(* CoDeSys 2.3.9.41 project: advance.pro *)
(* Libraries: UNM.lib 14.2.06 12:27:08, SmsOwenLib.lib 5.10.12 16:48:36, STANDARD.LIB 4.10.05 10:14:46, IECSFC.LIB 13.4.06 14:51:28, SYSLIBTIME.LIB 20.2.06 13:31:16, SYSTASKINFO.LIB 20.2.06 13:31:38, ANALYZATION.LIB 5.10.99 08:05:06, SYSLIBCALLBACK.LIB 20.2.06 13:31:08 *)

(* PLC configuration (modules and I/O channels)
Discrete input 8 bit [ID100] node 0, in %IB0 out %QB0 {Filtrationtime = 10; Filtrationtime = 10; Filtrationtime = 10; Filtrationtime = 10; Filtrationtime = 10; Filtrationtime = 10; Filtrationtime = 10; Filtrationtime = 10; Visibility = No; PinCount = 8; WatchDogPeriod = 1000; PollPeriod = 1}
  AT %IB0.0 [ByteInput] 8 discrete inputs
Discrete output 2 bit [ID101] node 1, in %IB1 out %QB1 {PinCount = 2; SafeValueBool = FALSE; SafeValueBool = FALSE; Visibility = No}
  pmp1 AT %QX1.0 [BitOutput] First
  pmp2 AT %QX1.1 [BitOutput] Second
Discrete output 2 bit [ID101] node 2, in %IB2 out %QB2 {PinCount = 2; SafeValueBool = FALSE; SafeValueBool = FALSE; Visibility = No}
  pmp3 AT %QX2.0 [BitOutput] First
  pmp4 AT %QX2.1 [BitOutput] Second
Discrete output 2 bit [ID101] node 3, in %IB3 out %QB3 {PinCount = 2; SafeValueBool = FALSE; SafeValueBool = FALSE; Visibility = No}
  AT %QX3.0 [BitOutput] First
  AT %QX3.1 [BitOutput] Second
Discrete output 2 bit [ID101] node 4, in %IB4 out %QB4 {PinCount = 2; SafeValueBool = FALSE; SafeValueBool = FALSE; Visibility = No}
  AT %QX4.0 [BitOutput] First
  AT %QX4.1 [BitOutput] Second
Discrete output 2 bit [ID101] node 5, in %IB5 out %QB5 {PinCount = 2; SafeValueBool = FALSE; SafeValueBool = FALSE; Visibility = No}
  AT %QX5.0 [BitOutput] First
  AT %QX5.1 [BitOutput] Second
Discrete output 2 bit [ID101] node 6, in %IB6 out %QB6 {PinCount = 2; SafeValueBool = FALSE; SafeValueBool = FALSE; Visibility = No}
  AT %QX6.0 [BitOutput] First
  AT %QX6.1 [BitOutput] Second
Special output [ID104] node 7, in %IB7 out %QB7 {Visibility = No; PinCount = 1}
  AT %QX7.0 [BitOutput] Special output
RS-232 [COM2_USART] node 0, in %IB8.0 out %QB8.0 {CommunicationSpeed = 9600; Parity = NO PARITY CHECK; BitLength = 8 bits; StopLength = One stop bit; InterfaceType = RS232; FrameOriented = ASCII; Timeout = 0; Visibility = No}
*)

(* Global variable list: Global_Variables *)
VAR_GLOBAL

	SMS_ID  : WORD;

END_VAR

(* POU PLC_PRG, ST *)
PROGRAM PLC_PRG
VAR
    startTimer, waitBeforeStartPmp2, waitBeforeStartPmp3, waitBeforeStartPmp4 : TON;
    letsGo : BOOL;
    letsStop : BOOL;
    stopTimer,waitBeforeStopPmp3,  waitBeforeStopPmp2, waitBeforeStopPmp1 : TON;
    startBreak, pmp2break, pmp3break, pmp4break : BOOL;

END_VAR
Process;

SMS;
END_PROGRAM
ACTION Process:
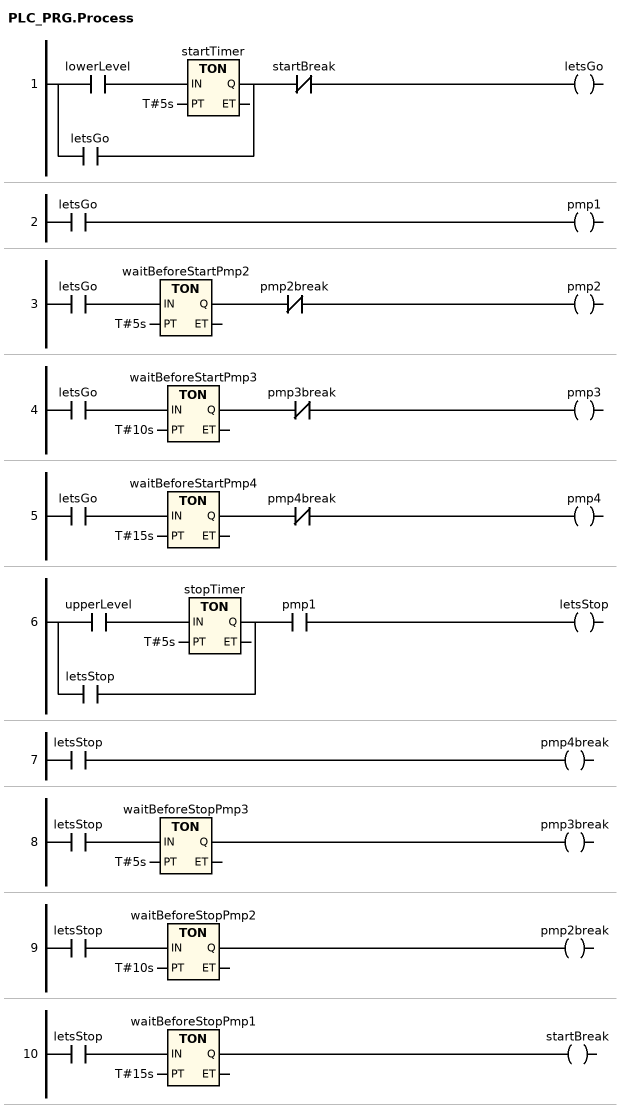
_LD_ (* Ladder Diagram *)
NETWORK 1
	{ [lowerLevel] - startTimer:TON(IN: *, PT: T#5s) | [letsGo] } - [/startBreak] --- (letsGo)
NETWORK 2
	[letsGo] --- (pmp1)
NETWORK 3
	[letsGo] - waitBeforeStartPmp2:TON(IN: *, PT: T#5s) - [/pmp2break] --- (pmp2)
NETWORK 4
	[letsGo] - waitBeforeStartPmp3:TON(IN: *, PT: T#10s) - [/pmp3break] --- (pmp3)
NETWORK 5
	[letsGo] - waitBeforeStartPmp4:TON(IN: *, PT: T#15s) - [/pmp4break] --- (pmp4)
NETWORK 6
	{ [upperLevel] - stopTimer:TON(IN: *, PT: T#5s) | [letsStop] } - [pmp1] --- (letsStop)
NETWORK 7
	[letsStop] --- (pmp4break)
NETWORK 8
	[letsStop] - waitBeforeStopPmp3:TON(IN: *, PT: T#5s) --- (pmp3break)
NETWORK 9
	[letsStop] - waitBeforeStopPmp2:TON(IN: *, PT: T#10s) --- (pmp2break)
NETWORK 10
	[letsStop] - waitBeforeStopPmp1:TON(IN: *, PT: T#15s) --- (startBreak)
_END_LD_
(* the same logic as Structured Text *)
(* Network 1 *)
startTimer(IN := lowerLevel, PT := T#5s);
letsGo := (startTimer.Q OR letsGo) AND NOT startBreak;
(* Network 2 *)
pmp1 := letsGo;
(* Network 3 *)
waitBeforeStartPmp2(IN := letsGo, PT := T#5s);
pmp2 := waitBeforeStartPmp2.Q AND NOT pmp2break;
(* Network 4 *)
waitBeforeStartPmp3(IN := letsGo, PT := T#10s);
pmp3 := waitBeforeStartPmp3.Q AND NOT pmp3break;
(* Network 5 *)
waitBeforeStartPmp4(IN := letsGo, PT := T#15s);
pmp4 := waitBeforeStartPmp4.Q AND NOT pmp4break;
(* Network 6 *)
stopTimer(IN := upperLevel, PT := T#5s);
letsStop := (stopTimer.Q OR letsStop) AND pmp1;
(* Network 7 *)
pmp4break := letsStop;
(* Network 8 *)
waitBeforeStopPmp3(IN := letsStop, PT := T#5s);
pmp3break := waitBeforeStopPmp3.Q;
(* Network 9 *)
waitBeforeStopPmp2(IN := letsStop, PT := T#10s);
pmp2break := waitBeforeStopPmp2.Q;
(* Network 10 *)
waitBeforeStopPmp1(IN := letsStop, PT := T#15s);
startBreak := waitBeforeStopPmp1.Q;
END_ACTION

(* POU SMS, ST *)
PROGRAM SMS
VAR
	Com		: OpenPort;
	cfg		       : FB_SMS_CFG;
	sms		: FB_SMS_SR;
	sl			: FB_SMS_SL;
	cfg_ok		: BOOL := FALSE;
	sendSMS  : BOOL := FALSE;
	ready		: BOOL;
	DevNum	: WORD := 0;
	openModemPort : BOOL := FALSE;
	port_ok      : BOOL := FALSE;
	errCode     : BYTE;
	errBool      : BOOL;

	sendText   : STRING(70);
	listNum	: ARRAY [0..1] OF STRING(20);
	sended     : BOOL;

	senderErrCode : BYTE;
	timeOut : TON;

	lock1, lock2, lock3, lock4 : BOOL := FALSE;

	RESERVE_1: BOOL;
	RESERVE_2: BOOL;
END_VAR
Inputs;
SelectNumber;

IF SMS_ID > 0 THEN
	Select;
	openModemPort := TRUE;
	sendSMS := TRUE;
ELSE
	openModemPort := FALSE;
	sendSMS := FALSE;
END_IF;

Configure;

IF ( cfg_ok=TRUE ) AND ( errBool=FALSE ) THEN
	ready := TRUE;
ELSE
	ready := FALSE;
END_IF;

Send;

IF sended THEN
	SMS_ID := 0;
	sendSMS := FALSE;
END_IF;

TimeoutSMS;
END_PROGRAM
ACTION Configure:
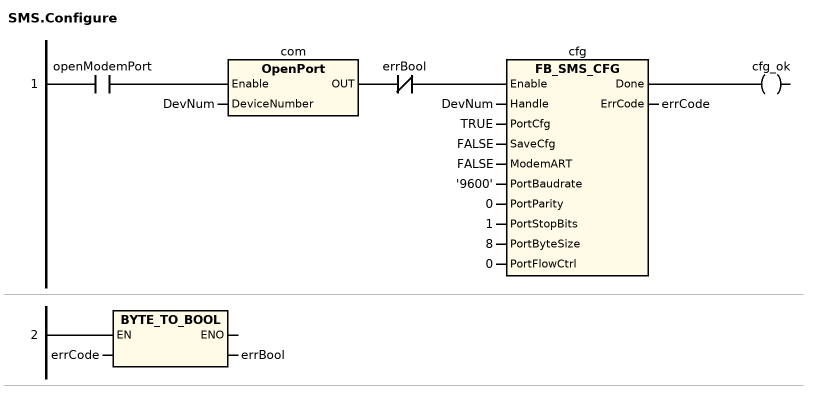
_LD_ (* Ladder Diagram *)
NETWORK 1
	[openModemPort] - com:OpenPort(Enable: *, DeviceNumber: DevNum) - [/errBool] - cfg:FB_SMS_CFG(Enable: *, Handle: DevNum, PortCfg: TRUE, SaveCfg: FALSE, ModemART: FALSE, PortBaudrate: '9600', PortParity: 0, PortStopBits: 1, PortByteSize: 8, PortFlowCtrl: 0, ErrCode => errCode) --- (cfg_ok)
NETWORK 2
	*
		EN --- BYTE_TO_BOOL(errCode) => errBool
_END_LD_
(* the same logic as Structured Text *)
(* Network 1 *)
com(Enable := openModemPort, DeviceNumber := DevNum);
cfg(Enable := com.OUT AND NOT errBool, Handle := DevNum, PortCfg := TRUE, SaveCfg := FALSE, ModemART := FALSE, PortBaudrate := '9600', PortParity := 0, PortStopBits := 1, PortByteSize := 8, PortFlowCtrl := 0);
errCode := cfg.ErrCode;
cfg_ok := cfg.Done;
(* Network 2 *)
errBool := BYTE_TO_BOOL(errCode);
END_ACTION
ACTION Inputs:
IF SMS_ID = 0 THEN
	IF upperLevel AND lock1=FALSE THEN
		SMS_ID := 1;
		lock1 := TRUE;
	END_IF;
	IF lowerLevel AND lock2=FALSE THEN
		SMS_ID := 2;
		lock2 := TRUE;
	END_IF;
	IF RESERVE_1 AND lock3=FALSE THEN
		SMS_ID := 4;
		lock3 := TRUE;
	END_IF;
	IF RESERVE_2 AND lock4=FALSE THEN
		SMS_ID := 8;
		lock4 := TRUE;
	END_IF;
END_IF;

IF upperLevel=FALSE THEN
	lock1 := FALSE;
END_IF;
IF lowerLevel=FALSE THEN
	lock2 := FALSE;
END_IF;
IF RESERVE_1=FALSE THEN
	lock3 := FALSE;
END_IF;
IF RESERVE_2=FALSE THEN
	lock4 := FALSE;
END_IF;
END_ACTION
ACTION Select:
IF SMS_ID.0 THEN
	sendText := 'Верхний уровень';
END_IF;

IF SMS_ID.1 THEN
	sendText := 'Нижний уровень';
END_IF;

IF SMS_ID.2 THEN
	sendText := 'reserve';
END_IF;

IF SMS_ID.3 THEN
	sendText := 'reserve';
END_IF;
END_ACTION
ACTION SelectNumber:
listNum[0] := '79123526879';

(* in work
listNum[0] := '79225418000';
listNum[1] := '79225306922';
*)
(*
listNum[0] := '79123526879';
listNum[1] := '79878552088';
*)
END_ACTION
ACTION Send:
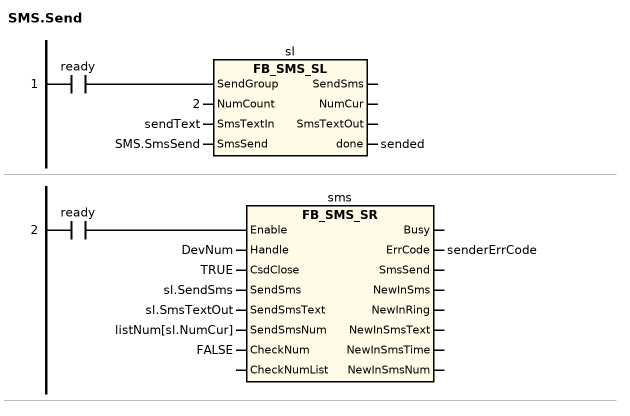
_LD_ (* Ladder Diagram *)
NETWORK 1
	[ready] - sl:FB_SMS_SL(SendGroup: *, NumCount: 2, SmsTextIn: sendText, SmsSend: SMS.SmsSend, done => sended)
NETWORK 2
	[ready] - sms:FB_SMS_SR(Enable: *, Handle: DevNum, CsdClose: TRUE, SendSms: sl.SendSms, SendSmsText: sl.SmsTextOut, SendSmsNum: listNum[sl.NumCur], CheckNum: FALSE, CheckNumList: , ErrCode => senderErrCode)
_END_LD_
(* the same logic as Structured Text *)
(* Network 1 *)
sl(SendGroup := ready, NumCount := 2, SmsTextIn := sendText, SmsSend := SMS.SmsSend);
sended := sl.done;
(* Network 2: see the listing above *)
END_ACTION
ACTION TimeoutSMS:
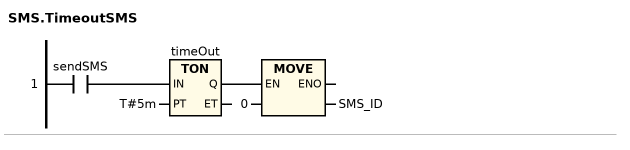
_LD_ (* Ladder Diagram *)
NETWORK 1
	[sendSMS] - timeOut:TON(IN: *, PT: T#5m)
		EN --- MOVE(0) => SMS_ID
_END_LD_
(* the same logic as Structured Text *)
(* Network 1 *)
timeOut(IN := sendSMS, PT := T#5m);
IF timeOut.Q THEN
	SMS_ID := 0;
END_IF;
END_ACTION
